(* IEC 61131-3 sources: controlforge-structured-text/manual-tests/completion, 4 files *)

(* ---- completion.st ---- *)
FUNCTION_BLOCK FB_TestMotor
VAR_INPUT
    enable : BOOL;
    speed : REAL;
END_VAR
VAR_OUTPUT
    running : BOOL;
    actual_speed : REAL;
END_VAR
END_FUNCTION_BLOCK

PROGRAM TestCompletion
VAR
    motor : FB_TestMotor;
    counter : INT := 0;
    temperature : REAL := 25.5;
END_VAR
// Press Ctrl+Space here to test completion
// You should see:
// - Keywords: IF, WHILE, FOR, etc.
// - Data types: BOOL, INT, REAL, etc.
// - Function blocks: TON, CTU, FB_TestMotor, etc.
// - Variables: motor, counter, temperature

END_PROGRAM

(* ---- lsp-stage2.st ---- *)
// Enhanced test file for Stage 2 LSP functionality
// Tests: Functions, Function Blocks, Programs, and various VAR sections

// Global variables
VAR_GLOBAL
    g_SystemRunning : BOOL := TRUE;
    g_EmergencyStop : BOOL := FALSE;
    g_MainCounter : INT := 0;
END_VAR

// Custom function with parameters
FUNCTION CalculateAverage : REAL
VAR_INPUT
    value1 : REAL;
    value2 : REAL;
    value3 : REAL;
END_VAR
VAR
    sum : REAL;
END_VAR

sum := value1 + value2 + value3;
CalculateAverage := sum / 3.0;

END_FUNCTION

// Custom function block
FUNCTION_BLOCK FB_PIDController
VAR_INPUT
    setpoint : REAL;
    processValue : REAL;
    kP : REAL := 1.0;
    kI : REAL := 0.1;
    kD : REAL := 0.01;
END_VAR
VAR_OUTPUT
    output : REAL;
    error : REAL;
END_VAR
VAR
    integral : REAL;
    lastError : REAL;
    derivative : REAL;
END_VAR

// PID calculation
error := setpoint - processValue;
integral := integral + error;
derivative := error - lastError;
output := kP * error + kI * integral + kD * derivative;
lastError := error;

END_FUNCTION_BLOCK

// Main program
PROGRAM MainControl
VAR
    // Standard function block instances
    mainTimer : TON;
    emergencyTrigger : R_TRIG;
    productCounter : CTU;

    // Custom function block instance
    temperatureController : FB_PIDController;

    // Local variables
    currentTemp : REAL;
    targetTemp : REAL := 75.5;
    timerRunning : BOOL;
    cycleCount : INT;
END_VAR

// --- MANUAL TEST INSTRUCTIONS ---
//
// 1. STANDARD FB CALL PARAMETERS
//    - Delete args from "mainTimer(...)" below, type "mainTimer(" and pause
//    - Expected: IN :=, PT := auto-suggested (TON inputs)
//    - Same for "emergencyTrigger(" → CLK :=
//    - Same for "productCounter(" → CU :=, R :=, PV :=

// 2. CUSTOM FB CALL PARAMETERS
//    - Delete args from "temperatureController(...)" below, type "temperatureController(" and pause
//    - Expected: setpoint :=, processValue :=, kP :=, kI :=, kD :=

// 3. MEMBER ACCESS ON STANDARD FB
//    - Place cursor after "mainTimer." on the timerRunning line and press Ctrl+Space
//    - Expected: IN, PT, Q, ET
//    - Place cursor after "productCounter." on the cycleCount line
//    - Expected: CU, R, PV, Q, CV

// 4. MEMBER ACCESS ON CUSTOM FB
//    - Type "temperatureController." somewhere in the body and press Ctrl+Space
//    - Expected: setpoint, processValue, kP, kI, kD, output, error

// 5. CROSS-POU FUNCTION CALL COMPLETION
//    - On a blank line type "Calc" and press Ctrl+Space
//    - Expected: CalculateAverage appears

// 6. GLOBAL VARIABLE COMPLETION
//    - On a blank line type "g_" and press Ctrl+Space
//    - Expected: g_SystemRunning, g_EmergencyStop, g_MainCounter

// Timer logic
mainTimer(IN := g_SystemRunning, PT := T#10s);
timerRunning := mainTimer.Q;

// Emergency stop detection
emergencyTrigger(CLK := g_EmergencyStop);

// Counter logic
productCounter(CU := timerRunning, R := emergencyTrigger.Q, PV := 100);
cycleCount := productCounter.CV;

// PID temperature control
temperatureController(
    setpoint := targetTemp,
    processValue := currentTemp,
    kP := 2.5,
    kI := 0.8,
    kD := 0.15
);

// Function call example
IF cycleCount > 50 THEN
    targetTemp := CalculateAverage(75.0, 80.0, 70.0);
END_IF

// Global variable usage
g_MainCounter := cycleCount;

END_PROGRAM

(* ---- instance-members.st ---- *)
PROGRAM TestInstanceCompletion
VAR
    // Timer instances - should show IN, PT, Q, ET when typing instanceName.
    pulseTimer : TP;
    onDelayTimer : TON;
    offDelayTimer : TOF;

    // Counter instances - CTU/CTD show Q and CV, CTUD shows QU, QD, CV
    upCounter : CTU;
    downCounter : CTD;
    upDownCounter : CTUD;

    // Edge trigger instances - should show CLK, Q when typing instanceName.
    risingEdge : R_TRIG;
    fallingEdge : F_TRIG;

    // Bistable instances - should show S/R1/Q1 or S1/R/Q1
    setReset : RS;
    resetSet : SR;

    // Test variables
    triggerSignal : BOOL := FALSE;
    resetSignal : BOOL := FALSE;
    counterValue : INT;
    timerOutput : BOOL;
END_VAR

// Manual test instructions:
// 1. Type "pulseTimer." + Ctrl+Space → should show IN, PT, Q, ET
// 2. Type "upCounter." + Ctrl+Space → should show CU, R, PV, Q, CV
// 3. Type "upDownCounter." + Ctrl+Space → should show CU, CD, R, LD, PV, QU, QD, CV
// 4. Type "risingEdge." + Ctrl+Space → should show CLK, Q
// 5. Type "setReset." + Ctrl+Space → should show S, R1, Q1

// Example usage:
pulseTimer(IN := triggerSignal, PT := T#2s);
timerOutput := pulseTimer.Q;

upCounter(CU := triggerSignal, R := resetSignal, PV := 100);
counterValue := upCounter.CV;

IF upCounter.CV >= 10 THEN
    resetSignal := TRUE;
END_IF

END_PROGRAM

(* ---- lsp.st ---- *)
PROGRAM TestProgram
VAR
    myTimer : TON;
    counter : INT;
    isActive : BOOL;
    temperature : REAL;
END_VAR

// --- MANUAL TEST INSTRUCTIONS ---
//
// 1. MEMBER ACCESS (dot completion)
//    - Place cursor after "myTimer." on line below and press Ctrl+Space
//    - Expected: IN, PT, Q, ET
myTimer(IN := isActive, PT := T#5s);

// 2. FB CALL PARAMETERS (trigger on open paren)
//    - Delete the contents of the call above, type "myTimer(" and pause
//    - Expected: IN :=, PT := auto-suggested
//    - Type a param e.g. "IN := isActive, " then press Ctrl+Space again
//    - Expected: PT := still suggested

// 3. VARIABLE COMPLETION
//    - On a blank line in the body, type "co" and press Ctrl+Space
//    - Expected: counter appears in list

// 4. KEYWORD COMPLETION
//    - On a blank line, type "IF" and press Ctrl+Space
//    - Expected: IF keyword in list

// 5. DATA TYPE COMPLETION
//    - On a blank line in VAR, type "IN" and press Ctrl+Space
//    - Expected: INT, LINT, DINT, USINT, UINT, UDINT, ULINT visible
counter := counter + 1;
temperature := 25.5;

IF myTimer.Q THEN
    isActive := FALSE;
END_IF

END_PROGRAM
